Staubli VAL3: setEventAndWait.pgx

public program setEventAndWait(num x_nCamID (dimensions=1), num x_nEvent (dimensions=1), bool& x_bError[] (dimensions=1))
begin
  //-----------------------------------------------------------------------
  //Header begin
  //Description of program
  //  Set event and wait until spreadsheet has been updated
  //
  //Input parameters
  //  num x_nCamID :
  //    role : camera's ID
  //  num x_nEvent  :
  //    role : The Event code to set
  //    possible values : (0 to 7), Specifies a soft trigger (Soft 0, Soft 1, ... Soft 7).
  //
  //Output parameters
  //  bool x_bError :
  //    role : returns true if an error occurred and false otherwise
  //
  //Examples
  //  call setEventAndWait(nCamID,nEvent,l_bError)
  //
  //History
  //  Creation : 19-05-08 - f.Rob
  //Header end
  //-----------------------------------------------------------------------

  nProgram[x_nCamID]=7
  call sendCommand(x_nCamID,"SW"+toString("0.0",x_nEvent),x_bError)
end
